PROGRAM POU_1
VAR
	
	objectDetected : BOOL := FALSE;

	blackObject : BOOL := FALSE;	
	redObject : BOOL := FALSE;
	
	motorOn : BOOL := FALSE;
	actuatorMove : BOOL := FALSE;
	
	objectSorted : BOOL := FALSE;
	
	startTimer : BOOL := FALSE;
	TON_0 : TON;	

END_VAR

TON_0(IN := startTimer, PT := T#5S);

IF objectDetected = TRUE THEN
	
	objectSorted := FALSE;
	
	IF redObject = TRUE THEN
		actuatorMove := TRUE;
	END_IF	

	startTimer := TRUE;
	motorOn := TRUE;

END_IF

IF TON_0.ET > T#1S THEN	
	
	motorOn := FALSE;
	startTimer := FALSE;
	actuatorMove := FALSE;
	
	objectSorted := TRUE;
	
END_IF

END_PROGRAM

(* stored: Version 1.1.0.1, ProductVersion 3.1.4024.3
   POU POU_1: Id {0092da42-47c0-4849-9c55-1c574ee8f141}, SpecialFunc None *)
